(* IEC 61131-3 sources: AXOpen/src/showcase/app/src/ComponentsRexrothTightening/Documentation, 1 file *)

(* ---- Component_1.st ---- *)
USING AXOpen.Core;
NAMESPACE AXOpen.Components.Rexroth.Tightening
    {S7.extern=ReadWrite}
    CLASS Component_1 EXTENDS AXOpen.Core.AxoObject
        //<ComponentDeclaration>
        VAR PUBLIC
            ExampleComponent : AXOpen.Components.Rexroth.Tightening.Axo_CS351_compact;
        END_VAR
        //</ComponentDeclaration>

        //<InitializationArgumentsDeclaration>
        VAR PUBLIC
            {#ix-set:AttributeName = "<#Activate manual control#>"}
            ActivateManualControl : BOOL;
        END_VAR
        //</InitializationArgumentsDeclaration>

        METHOD PUBLIC OVERRIDE Run
            VAR_INPUT
                inParent : IAxoObject;
            END_VAR

            SUPER.Run(inParent);

            IF ActivateManualControl THEN
                ExampleComponent.ActivateManualControl();
            END_IF;

            //<Initialization>
            ExampleComponent.Run(inParent := THIS , hwID:= AXOpen.Showcase.HwIdentifiers#rexroth_cs351_HwID);
            //</Initialization>

            THIS.UseInSequencer();
        END_METHOD

        //<Usage>
        VAR PUBLIC
            Sequencer : AxoSequencer;
            Steps : ARRAY[0..30] OF AXOpen.Core.AxoStep;
        END_VAR

        METHOD PRIVATE UseInSequencer
            IF Sequencer.GetContext().OpenCycleCount() = ULINT#0 THEN
                Sequencer.SequenceMode := eAxoSequenceMode#RunOnce;
            END_IF;

            Sequencer.Run(THIS);
            Sequencer.Open();

            IF(Steps[0].Execute(Sequencer, 'Disable')) THEN
                IF(ExampleComponent.Disable().IsDone()) THEN
                    Sequencer.MoveNext();
                END_IF;
            END_IF;

            IF(Steps[1].Execute(Sequencer, 'Enable')) THEN
                IF(ExampleComponent.Enable().IsDone()) THEN
                    Sequencer.MoveNext();
                END_IF;
            END_IF;

            IF(Steps[2].Execute(Sequencer, 'DisableClockwise')) THEN
                IF(ExampleComponent.DisableClockwise().IsDone()) THEN
                    Sequencer.MoveNext();
                END_IF;
            END_IF;

            IF(Steps[3].Execute(Sequencer, 'EnableClockwise')) THEN
                IF(ExampleComponent.EnableClockwise().IsDone()) THEN
                    Sequencer.MoveNext();
                END_IF;
            END_IF;

            IF(Steps[4].Execute(Sequencer, 'DisableCounterClockwise')) THEN
                IF(ExampleComponent.DisableCounterClockwise().IsDone()) THEN
                    Sequencer.MoveNext();
                END_IF;
            END_IF;

            IF(Steps[5].Execute(Sequencer, 'EnableCounterClockwise')) THEN
                IF(ExampleComponent.EnableCounterClockwise().IsDone()) THEN
                    Sequencer.MoveNext();
                END_IF;
            END_IF;

            IF(Steps[6].Execute(Sequencer, 'ResetFault')) THEN
                IF(ExampleComponent.ResetFault().IsDone()) THEN
                    Sequencer.MoveNext();
                END_IF;
            END_IF;

            IF(Steps[7].Execute(Sequencer, 'ResetResults')) THEN
                IF(ExampleComponent.ResetResults().IsDone()) THEN
                    Sequencer.MoveNext();
                END_IF;
            END_IF;

            IF(Steps[8].Execute(Sequencer, 'SetScrewingProgram')) THEN
                IF(ExampleComponent.SetScrewingProgram(BYTE#5).IsDone()) THEN
                    Sequencer.MoveNext();
                END_IF;
            END_IF;

            IF(Steps[9].Execute(Sequencer, 'GetScrewingResults')) THEN
                IF(ExampleComponent.GetScrewingResults().IsDone()) THEN
                    Sequencer.MoveNext();
                END_IF;
            END_IF;

            IF(Steps[10].Execute(Sequencer, 'ScrewClockwise')) THEN
                IF(ExampleComponent.ScrewClockwise(TRUE).IsDone()) THEN
                    Sequencer.MoveNext();
                END_IF;
            END_IF;

            IF(Steps[11].Execute(Sequencer, 'ScrewCounterClockwise')) THEN
                IF(ExampleComponent.ScrewCounterClockwise(TRUE).IsDone()) THEN
                    Sequencer.MoveNext();
                END_IF;
            END_IF;

            IF(Steps[12].Execute(Sequencer, 'RunAutomat')) THEN
                IF(ExampleComponent.RunAutomat(BYTE#5,'test',TRUE).IsDone()) THEN
                    Sequencer.MoveNext();
                END_IF;
            END_IF;

            IF(Steps[13].Execute(Sequencer, 'Restore')) THEN
                ExampleComponent.Restore();
                Sequencer.CompleteSequence();
            END_IF;

        END_METHOD

        //</Usage>
    END_CLASS
END_NAMESPACE
